{attribute 'qualified_only'}
{attribute 'strict'}
TYPE E_DoorState :
(
	CLOSED := 0,
	OPENING := 1,
	OPEN := 2,
	CLOSING := 3
) INT;
END_TYPE

(* stored: Version 1.1.0.1
   DUT E_DoorState: Id {f5fb6cd7-5a1e-4cb8-8c17-64673322d861} *)
